// TIA Portal V20 export
// export: Created 2025-12-01T14:57:09.2054012Z, ExportSetting None, DisplayName Totally Integrated Automation Portal, DisplayVersion V20 Update 3, DisplayName TIA Portal Openness, DisplayVersion V20 Update 3, DisplayName TIA Portal Version Control Interface, DisplayVersion V20 Update 3, DisplayName STEP 7 Professional, DisplayVersion V20 Update 3, DisplayName STEP 7 Safety, DisplayVersion V20 Update 2, DisplayName WinCC Basic/Comfort/Advanced, DisplayVersion V20 Update 3, DisplayName WinCC Professional, DisplayVersion V20 Update 3, DisplayName WinCC Unified, DisplayVersion V20 Update 3
FUNCTION "FC834_GestorMaquinaSimple" : Void   // FC834, LAD
TITLE = Tracking de la Maquina Base
{ S7_Optimized_Access := 'FALSE' }
AUTHOR : TRACKING
NAME : 20160525
VERSION : 3.1
// - Inicializar
// - Recoger datos necesarios del Sistema
// 
// - Dispositivo Maquina
//   + Gestion de Estado
//   + Gestion de Control de Reset
//   + Gestion de Control de Paro Blando
//   + Gestion de Control de Errores
// 
// - Operaciones propias de la Maquina
// 
// - Cierre de protocolo de la Maquina
// - Actualizar datos del Sistema
// stored: AutoNumber false, SetENOAutomatically false
   VAR_INPUT
      DB_VIMaquina : DB_ANY;   // DB de la Maquina
      EstadoZonaMesa : "EstadoZona";   // Estado de la Zona Mesa Asociada a la Mesa
      NumMaquina : UInt;   // Numero de la Maquina
      RearmeError : Bool;   // Rearme de Errores Adicionales
      ManualReset : Bool;   // Resetear la Maquina desde el exterior
      FinReset : Bool;   // Reset Finalizado del VI Maquina
      ManualParoBlando : Bool;   // Paro Blando de la Mauina desde el exterior
      FinParoBlando : Bool;   // Paro Blando Finalizado del VI Maquina
   END_VAR
   VAR_TEMP
      PunteroDBVIMaquina : Any;
      P_EstadoVI : DWord;
      PunteroDBTMP : DWord;
      DBEstadoVI : Word;
      CodigoErrorMesa : UDInt;   // Error (Código) de la Mesa (Dispositivo)
      NumeroErrorVI : UInt;
      Maquina : UInt;   // Numero de Maquina dentro del PLC
      ByteTMP : Byte;
      ReturnValor : Int;
      TMPFinReset_NOK : Bool;
      TMPFinParoBlando_NOK : Bool;
      FlancoAuto : Bool;
      FlancoManual : Bool;
      FlancoMarcha : Bool;
      FlancoParo : Bool;
      FlancoReset : Bool;
      FlancoParoBlando : Bool;
      FinResetTMP : Bool;
      FinParoBlandoTMP : Bool;
   END_VAR
BEGIN

NETWORK
TITLE = Inicializar
/////////////////////////////////////////////////////////////////////////////
// --- Inicializar las Variables

      L     #NumMaquina;
      T     #Maquina;


/////////////////////////////////////////////////////////////////////////////
// --- Estado Mesa - Salida Inicializar a cero - Zona

      L     0;  // Que rellenar en el DB
      T     #ByteTMP;

      CALL  FILL
      ( BVAL    := #ByteTMP,
        RET_VAL := #ReturnValor,
        BLK     := "DB903_Estado_ZonaMaquina".EstadoMaquina[#Maquina]
      );  // Reseteo el la zona temp



NETWORK
TITLE = Gestion del Estado de la Maquina - Inicial
/////////////////////////////////////////////////////////////////////////////
// --- Flancos de los estados de la Maquina

      SET;
      A     #EstadoZonaMesa.Automatico_CBx;
      FP    "DB832_Maquinas".Maquinas[#Maquina].Memorias.MFL_Auto;  // Memo Automatico
      =     #FlancoAuto;

      SET;
      A     #EstadoZonaMesa.Manual_CBx;
      FP    "DB832_Maquinas".Maquinas[#Maquina].Memorias.MFL_Manual;  // Memo Manual
      =     #FlancoManual;

      SET;
      A     #EstadoZonaMesa.Marcha_CBx;
      FP    "DB832_Maquinas".Maquinas[#Maquina].Memorias.MFL_Marcha;  // Memo Marcha
      =     #FlancoMarcha;

      SET;
      A     #EstadoZonaMesa.Paro_CBx;
      FP    "DB832_Maquinas".Maquinas[#Maquina].Memorias.MFL_Paro;  // Memo Paro
      =     #FlancoParo;



NETWORK
TITLE = ---- Automatico, Manual
/////////////////////////////////////////////////////////////////////////////
// --- Estado de la Maquina
// --- Nota: Si cambia Auto/Remoto/Manual se pasa a Paro
// --- Nota: Si hay Marcha solo si esta en Automatico o Remoto
// ---       nunca en Manual

/////////////////////////////////////////////////////////////////////////////
// --- Maquina en Automatico (Estado: Automatico y Paro)
// --- Condicion: si la Zona Mesa esta en Automatico
      SET;
      A(;
      O     #FlancoAuto;  // Automatico de la Zona Mesa
      O     "DB841_Recepcion".DispoMaquina[#Maquina].Protocolo.Automatico;  // Automatico de la Orden Maquina
      );
      A     #EstadoZonaMesa.Automatico_CBx;  // Condicion
      JCN   NoEsta_EstadoDeLlaveEnAutomatico;

      SET;
      S     "DB840_Emision".DispoMaquina[#Maquina].Protocolo.Automatico;  // Poner en Automatico
      R     "DB840_Emision".DispoMaquina[#Maquina].Protocolo.Manual;

      JU    Final_EstadoDeLLave;

NoEsta_EstadoDeLlaveEnAutomatico:NOP   0;


/////////////////////////////////////////////////////////////////////////////
// --- Maquina en Manual (Estado: Manual y Paro)
// --- Condicion: Ninguna

      SET;
      A(;
      O     #FlancoManual;  // Manual de la Zona Mesa
      O     "DB841_Recepcion".DispoMaquina[#Maquina].Protocolo.Manual;  // Manual de la Orden Maquina
      );
      JCN   NoEsta_EstadoDeLlaveEnManual;

      SET;
      R     "DB840_Emision".DispoMaquina[#Maquina].Protocolo.Automatico;  // Poner en Manual
      S     "DB840_Emision".DispoMaquina[#Maquina].Protocolo.Manual;

      JU    Final_EstadoDeLLave;

NoEsta_EstadoDeLlaveEnManual:NOP   0;


/////////////////////////////////////////////////////////////////////////////
// --- Final Control de Llave de Mesa (En Automatico y En Manual)
Final_EstadoDeLLave:NOP   0;



NETWORK
TITLE = ---- Marcha, Paro
/////////////////////////////////////////////////////////////////////////////
// --- Maquina en Marcha
// --- Condicion: si esta la Maquina en Automatico o Remoto
// ---            si esta la Zona Mesa en Marcha

      SET;
      A(;
      O     #FlancoMarcha;  // Marcha de la Zona Mesa
      O     "DB841_Recepcion".DispoMaquina[#Maquina].Protocolo.Marcha;  // Marcha de la Orden Maquina
      );
      AN    #EstadoZonaMesa.Manual_CBx;  // Condiciones
      A     #EstadoZonaMesa.Marcha_CBx;

      AN    "DB840_Emision".DispoMaquina[#Maquina].Protocolo.Reset_Realizandose;
      JCN   NoEsta_EstadoDeMesaEnMarcha;

      SET;
      S     "DB840_Emision".DispoMaquina[#Maquina].Protocolo.Marcha;  // Poner en Marcha
      R     "DB840_Emision".DispoMaquina[#Maquina].Protocolo.Paro;
      R     "DB840_Emision".DispoMaquina[#Maquina].Protocolo.ParoBlando_Realizandose;  // Resetear Variables
      R     "DB840_Emision".DispoMaquina[#Maquina].Protocolo.ParoBlandoNOK;  // De Paro Blando
      R     "DB840_Emision".DispoMaquina[#Maquina].Protocolo.ParoBlandoOK;

      JU    Final_EstadoDeMesa;

NoEsta_EstadoDeMesaEnMarcha:NOP   0;


/////////////////////////////////////////////////////////////////////////////
// --- Maquina en Paro
// --- Condicion: Ninguna

      SET;
      A     #FlancoParo;  // Paro de la Zona Mesa
      O     "DB841_Recepcion".DispoMaquina[#Maquina].Protocolo.Paro;  // Paro de la Orden Maquina

      O     #FlancoAuto;  // Automatcio de la Zona Mesa
      O     #FlancoManual;  // Manual de la Zona Mesa

      O     "DB841_Recepcion".DispoMaquina[#Maquina].Protocolo.Automatico;  // Automatico de la Orden Maquina
      O     "DB841_Recepcion".DispoMaquina[#Maquina].Protocolo.Manual;  // Manual de la Orden Maquina

      JCN   NoEsta_EstadoDeMesaEnParo;

      SET;
      R     "DB840_Emision".DispoMaquina[#Maquina].Protocolo.Marcha;  // Poner en Paro
      S     "DB840_Emision".DispoMaquina[#Maquina].Protocolo.Paro;

NoEsta_EstadoDeMesaEnParo:NOP   0;


/////////////////////////////////////////////////////////////////////////////
// --- Final del control de Estado de Mesa (Marcha, Paro)
Final_EstadoDeMesa:NOP   0;




NETWORK
TITLE = Temporizador de Reset y Paro Blando NOK
/////////////////////////////////////////////////////////////////////////////
// --- Temporizador de Fin de Reset NOK

      CALL  "FC899_TMP"
      ( Temporizar     := "DB840_Emision".DispoMaquina[#Maquina].Protocolo.Reset_Realizandose,
        Valor_Tiempo   := "CTE_TMPEsperaFinReset",
        Base_tiempo_ms := 1000,
        Tiempo_OK      := #TMPFinReset_NOK,
        Valor_Actual   := "DB832_Maquinas".Maquinas[#Maquina].TMP_Reset
      );


/////////////////////////////////////////////////////////////////////////////
// --- Temporizador de Fin de ParoBlando NOK

      CALL  "FC899_TMP"
      ( Temporizar     := "DB840_Emision".DispoMaquina[#Maquina].Protocolo.ParoBlando_Realizandose,
        Valor_Tiempo   := "CTE_TMPEsperaFinReset",
        Base_tiempo_ms := 1000,
        Tiempo_OK      := #TMPFinParoBlando_NOK,
        Valor_Actual   := "DB832_Maquinas".Maquinas[#Maquina].TMP_ParoBlando
      );



NETWORK
TITLE = Gestion de Control de Reset
/////////////////////////////////////////////////////////////////////////////
// --- Flanco de Activacion de Reset

      SET;
      A     #EstadoZonaMesa.Resetear_CBx;  // Por la Zona Mesa
      O     #ManualReset;  // Manualmente (Exterior)
      O     "DB841_Recepcion".DispoMaquina[#Maquina].Protocolo.Reset;  // Por la Orden
      FP    "DB832_Maquinas".Maquinas[#Maquina].Memorias.MFL_Reset;  // Memo Reset
      =     #FlancoReset;

      SET;
      A     #FinReset;  // No hace caso si no hay Reset
      A     "DB904_Estado_Maquinas".EstadoVI[#Maquina].Fin_VI;
      A     "DB840_Emision".DispoMaquina[#Maquina].Protocolo.Reset_Realizandose;
      =     #FinResetTMP;

/////////////////////////////////////////////////////////////////////////////
// --- Activacion del Proceso de Reset

      SET;
      AN    #FlancoReset;
      JC    SistemaReset_Gestion;  // Hay que Realizar el Reset ?

      SET;
      A     "DB840_Emision".DispoMaquina[#Maquina].Protocolo.Marcha;
      JC    ResetImposible;


/////////////////////////////////////////////////////////////////////////////
// --- Se ha producido un Reset valido (Reseteo de las variables)

      SET;
      S     "DB840_Emision".DispoMaquina[#Maquina].Protocolo.Reset_Realizandose;  // Reseteando la Maquina
      R     "DB840_Emision".DispoMaquina[#Maquina].Protocolo.ParoBlando_Realizandose;  // Resetear Variables
      R     "DB840_Emision".DispoMaquina[#Maquina].Protocolo.ParoBlandoNOK;  // De Paro Blando
      R     "DB840_Emision".DispoMaquina[#Maquina].Protocolo.ParoBlandoOK;

      L     0;  // Reseteo el Status de Trabajo
      T     "DB832_Maquinas".Maquinas[#Maquina].MemoriaEstado;  // NuevoStatusTrabajo


/////////////////////////////////////////////////////////////////////////////
// --- Reseteo - DB del Vehiculo Inteligente

      OPN   #DB_VIMaquina;  // Abro el DB a resetear
      LAR1  P##PunteroDBVIMaquina;  // Preparar Puntero Any
      L     B#16#10;  // ID de Sintasis
      T     LB [AR1, P#0.0];
      L     B#16#2;  // Tipo de Datos
      T     LB [AR1, P#1.0];
      L     DBLG;  // Longitud del DB
      T     LW [AR1, P#2.0];
      L     DBNO;  // Numero de DB
      T     LW [AR1, P#4.0];
      L     0;
      SLW   3;
      T     LD [AR1, P#6.0];
      L     B#16#84;  // Indico el tipo DB
      T     LB [AR1, P#6.0];

      L     0;  // Que rellenar en el DB
      T     #ByteTMP;
      CALL  FILL
      ( BVAL    := #ByteTMP,
        RET_VAL := #ReturnValor,
        BLK     := #PunteroDBVIMaquina
      );  // Reseteo el DB


/////////////////////////////////////////////////////////////////////////////
// --- Reseteo - Estado del Vehiculo Inteligente

      L     0;  // Reseteo del Estado del VI
      T     #ByteTMP;
      CALL  FILL
      ( BVAL    := #ByteTMP,
        RET_VAL := #ReturnValor,
        BLK     := "DB904_Estado_Maquinas".EstadoVI[#Maquina]
      );


/////////////////////////////////////////////////////////////////////////////
// --- No hay más que resetar
      JU    SistemaReset_Gestion;


/////////////////////////////////////////////////////////////////////////////
// --- Reset Imposible

ResetImposible:NOP   0;
      SET;
      S     "DB840_Emision".DispoMaquina[#Maquina].Protocolo.ResetNOK;  // Activa del Bit Reset Imposible
      R     "DB840_Emision".DispoMaquina[#Maquina].Protocolo.ResetOK;  // Desactiva el Bit de Reset OK
      R     "DB840_Emision".DispoMaquina[#Maquina].Protocolo.Reset_Realizandose;

      JU    SistemaReset_Gestion;


/////////////////////////////////////////////////////////////////////////////
/////////////////////////////////////////////////////////////////////////////
/////////////////////////////////////////////////////////////////////////////
/////////////////////////////////////////////////////////////////////////////
// --- Gestion de Reset
SistemaReset_Gestion:NOP   0;
      SET;
      AN    "DB840_Emision".DispoMaquina[#Maquina].Protocolo.Reset_Realizandose;
      JC    SistemaReset_Fin;

      SET;
      AN    #EstadoZonaMesa.Resetear_CBx;  // Por la Zona
      AN    #EstadoZonaMesa.PerReset_CBx;
      AN    #ManualReset;  // Manualmente (Exterior)
      AN    "DB841_Recepcion".DispoMaquina[#Maquina].Protocolo.Reset;  // Por la Orden
      A     "DB841_Recepcion".DispoMaquina[#Maquina].Protocolo.EmiOK;  // Avisado el JdT ?
      JCN   SistemaReset_Continuar;


/////////////////////////////////////////////////////////////////////////////
// --- Reset Finalizazado
      SET;
      R     "DB840_Emision".DispoMaquina[#Maquina].Protocolo.Reset_Realizandose;


/////////////////////////////////////////////////////////////////////////////
// --- Continuar con el Reset
SistemaReset_Continuar:NOP   0;
      SET;
      A     #FinResetTMP;  // Fin de Reset del VI ?
      S     "DB840_Emision".DispoMaquina[#Maquina].Protocolo.ResetOK;  // Aviso de Fin de Reset


// --- Si no llega el Fin de Reset en un tiempo determinado
      SET;
      AN    #FinResetTMP;  // No, Fin de Reset del VI ?
      AN    "DB840_Emision".DispoMaquina[#Maquina].Protocolo.ResetOK;  // No, Aviso de Fin de Reset
      AN    "DB840_Emision".DispoMaquina[#Maquina].Protocolo.ResetNOK;  // No, Aviso de Fin de Reset
      A     #TMPFinReset_NOK;  // Se cumplido el tiempo de Espera
      A     "DB840_Emision".DispoMaquina[#Maquina].Protocolo.Reset_Realizandose;  // Reset Realizandose
      JC    ResetImposible;  // Activar reset imposible


/////////////////////////////////////////////////////////////////////////////
// --- Final de la Gestion de Reset
SistemaReset_Fin:NOP   0;
      SET;
      AN    "DB840_Emision".DispoMaquina[#Maquina].Protocolo.Reset_Realizandose;
      R     "DB840_Emision".DispoMaquina[#Maquina].Protocolo.ResetOK;  // No Aviso de Fin de Reset

      SET;
      A     "DB840_Emision".DispoMaquina[#Maquina].Protocolo.ResetNOK;
      A     "DB841_Recepcion".DispoMaquina[#Maquina].Protocolo.EmiOK;
      R     "DB840_Emision".DispoMaquina[#Maquina].Protocolo.ResetNOK;  // Desactivacion de Reset Imposible



NETWORK
TITLE = Gestion del Control de Paro Blando
// - Sistema de Paro Blando
//   * Flanco de Activacion del Paro Blando
//   * Activacion del proceso de Paro Blando
//   * Gestion del Paro Blando
/////////////////////////////////////////////////////////////////////////////
// --- Flanco de Activacion de Paro Blando

      SET;
      A     #EstadoZonaMesa.ParoBlando_CBx;  // Por la Zona Mesa
      O     #ManualParoBlando;  // Manualmente (Exterior)
      O     "DB841_Recepcion".DispoMaquina[#Maquina].Protocolo.ParoBlando;  // Por la Orden
      FP    "DB832_Maquinas".Maquinas[#Maquina].Memorias.MFL_ParoBlando;  // Memo Paro Blando - Pos: 22.7
      =     #FlancoParoBlando;

      SET;
      A     #FinParoBlando;  // No hace caso si no hay ParoBlando
      A     "DB904_Estado_Maquinas".EstadoVI[#Maquina].Paro_Blando;
      A     "DB840_Emision".DispoMaquina[#Maquina].Protocolo.ParoBlando_Realizandose;
      =     #FinParoBlandoTMP;


/////////////////////////////////////////////////////////////////////////////
// --- Activacion del Proceso de Paro Blando
      SET;
      AN    #FlancoParoBlando;
      JC    SistemaParoBlando_Gestion;  // Hay que Realizar el Paro Blando ?


/////////////////////////////////////////////////////////////////////////////
// --- Se ha producido un Paro Blando valido
      SET;
      S     "DB840_Emision".DispoMaquina[#Maquina].Protocolo.ParoBlando_Realizandose;  // Reseteando la Maquina

      JU    SistemaParoBlando_Gestion;


/////////////////////////////////////////////////////////////////////////////
// --- Paro Blando Imposible

ParoBlandoImposible:NOP   0;
      SET;
      S     "DB840_Emision".DispoMaquina[#Maquina].Protocolo.ParoBlandoNOK;  // Activacion de Paro Blando Imposible
      R     "DB840_Emision".DispoMaquina[#Maquina].Protocolo.ParoBlandoOK;  // DesActivacion de Paro Blando OK
      R     "DB840_Emision".DispoMaquina[#Maquina].Protocolo.ParoBlando_Realizandose;  // Acabado Paro Blando

      JU    SistemaParoBlando_Gestion;

/////////////////////////////////////////////////////////////////////////////
/////////////////////////////////////////////////////////////////////////////
/////////////////////////////////////////////////////////////////////////////
// --- Gestion de Paro Blando
SistemaParoBlando_Gestion:NOP   0;
      SET;
      AN    "DB840_Emision".DispoMaquina[#Maquina].Protocolo.ParoBlando_Realizandose;
      JC    SistemaParoBlando_Fin;

      SET;
      AN    #EstadoZonaMesa.ParoBlando_CBx;  // Por la Zona
      AN    #ManualParoBlando;  // Manualmente (Exterior)
      AN    "DB841_Recepcion".DispoMaquina[#Maquina].Protocolo.ParoBlando;  // Por la Orden
      A     "DB841_Recepcion".DispoMaquina[#Maquina].Protocolo.EmiOK;  // Avisado el JdT ?
      JCN   SistemaParoBlando_Continuar;


/////////////////////////////////////////////////////////////////////////////
/////////////////////////////////////////////////////////////////////////////
/////////////////////////////////////////////////////////////////////////////
// --- Paro Blando Finalizazado
      SET;
      R     "DB840_Emision".DispoMaquina[#Maquina].Protocolo.ParoBlando_Realizandose;


/////////////////////////////////////////////////////////////////////////////
/////////////////////////////////////////////////////////////////////////////
/////////////////////////////////////////////////////////////////////////////
// --- Continuar con el Reset
SistemaParoBlando_Continuar:NOP   0;
      SET;
      A     #FinParoBlandoTMP;  // Fin de Paro Blando del VI ?
      S     "DB840_Emision".DispoMaquina[#Maquina].Protocolo.ParoBlandoOK;  // Aviso de Fin de Paro Blando


// --- Si no llega el Fin de Paro Blando en un tiempo determinado
      SET;
      AN    #FinParoBlandoTMP;  // No, Fin de Paro Blando del VI ?
      AN    "DB840_Emision".DispoMaquina[#Maquina].Protocolo.ParoBlandoOK;  // No, Aviso de Fin de Paro Blando
      AN    "DB840_Emision".DispoMaquina[#Maquina].Protocolo.ParoBlandoNOK;  // No, Aviso de Fin de Paro Blando
      A     #TMPFinParoBlando_NOK;  // Se cumplido el tiempo de Espera
      A     "DB840_Emision".DispoMaquina[#Maquina].Protocolo.ParoBlando_Realizandose;  // Paro Blando Realizandose
      JC    ParoBlandoImposible;  // Activar Paro Blando imposible


/////////////////////////////////////////////////////////////////////////////
/////////////////////////////////////////////////////////////////////////////
/////////////////////////////////////////////////////////////////////////////
// --- Final de la Gestion de Reset
SistemaParoBlando_Fin:NOP   0;
      SET;
      AN    "DB840_Emision".DispoMaquina[#Maquina].Protocolo.ParoBlando_Realizandose;
      R     "DB840_Emision".DispoMaquina[#Maquina].Protocolo.ParoBlandoOK;  // No Aviso de Fin de Reset

      SET;
      A     "DB840_Emision".DispoMaquina[#Maquina].Protocolo.ParoBlandoNOK;
      A     "DB841_Recepcion".DispoMaquina[#Maquina].Protocolo.EmiOK;
      R     "DB840_Emision".DispoMaquina[#Maquina].Protocolo.ParoBlandoNOK;  // Desactivacion de Paro Blando Imposible



NETWORK
TITLE = Gestion de Control de Error de la Maquina
// - Calculo del Error de la Maquina
// - Rearme y Activacion del Error de la Maquina
/////////////////////////////////////////////////////////////////////////////
// --- Calculo del Error de la Mesa

      AN    "DB904_Estado_Maquinas".EstadoVI[#Maquina].Error_MAQx;
      JC    NoErrorEnMaquina;


/////////////////////////////////////////////////////////////////////////////
      L     #Maquina;  // Puntero al DB de Estado VI
      L     "CTE_Long_VIMaquina";  // Longitud de la UDT 20
      *D;
      SLD   3;
      T     #P_EstadoVI;

      L     "CTE_NDB_EstadoVIMaquina";  // DB de Estado VI
      T     #DBEstadoVI;

      L     #P_EstadoVI;  // Punteros
      L     P#2.0;
      +D;
      LAR2;
      T     #PunteroDBTMP;  // Offset dentro del DB

      OPN   DB [#DBEstadoVI];
Bucle_ErrorVI:NOP   0;
      A     DBX [AR2, P#0.0];
      JC    EncontradoErrorEnMaquina;

      +AR2  P#0.1;
      JU    Bucle_ErrorVI;


/////////////////////////////////////////////////////////////////////////////
// --- Con Error
EncontradoErrorEnMaquina:NOP   0;
      TAR2;
      L     #PunteroDBTMP;
      -D;
      L     51;
      +D;
      T     #NumeroErrorVI;
      T     "DB840_Emision".DispoMaquina[#Maquina].Error;

      L     #NumeroErrorVI;
      T     #CodigoErrorMesa;
      T     "DB861_FIFO_Errores".Maquinas[#Maquina];

      JU    FinGestion_Error;


/////////////////////////////////////////////////////////////////////////////
// --- Sin Error
NoErrorEnMaquina:NOP   0;
      L     0;
      T     #CodigoErrorMesa;
      T     "DB840_Emision".DispoMaquina[#Maquina].Error;
      T     "DB861_FIFO_Errores".Maquinas[#Maquina];

      JU    FinGestion_Error;


/////////////////////////////////////////////////////////////////////////////
// --- Rearme y Activacion del Error
FinGestion_Error:NOP   0;
      SET;
      A     #EstadoZonaMesa.Rearme_CBx;  // Por la Zona
      O     #RearmeError;  // Manualmente (Exterior)
      O     "DB841_Recepcion".DispoMaquina[#Maquina].Protocolo.Rearme;  // Por la Orden
      =     "DB903_Estado_ZonaMaquina".EstadoMaquina[#Maquina].Rearme_CBx;

      SET;
      A     "DB904_Estado_Maquinas".EstadoVI[#Maquina].Error_MAQx;
      =     "DB840_Emision".DispoMaquina[#Maquina].Protocolo.Error;  // Esta en Error el VI Maquina



REGION Network 9: Cierre del Protocolo de la Maquina
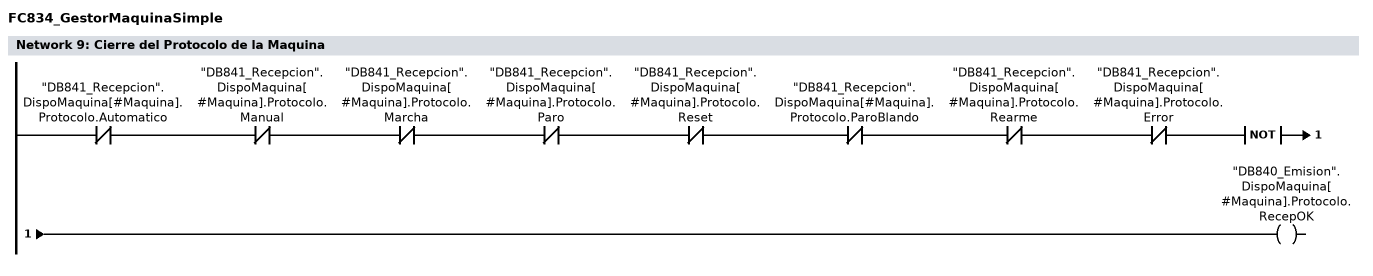
   RUNG wire#powerrail
      I_Contact( "DB841_Recepcion".DispoMaquina[#Maquina].Protocolo.Automatico )
      I_Contact( "DB841_Recepcion".DispoMaquina[#Maquina].Protocolo.Manual )
      I_Contact( "DB841_Recepcion".DispoMaquina[#Maquina].Protocolo.Marcha )
      I_Contact( "DB841_Recepcion".DispoMaquina[#Maquina].Protocolo.Paro )
      I_Contact( "DB841_Recepcion".DispoMaquina[#Maquina].Protocolo.Reset )
      I_Contact( "DB841_Recepcion".DispoMaquina[#Maquina].Protocolo.ParoBlando )
      I_Contact( "DB841_Recepcion".DispoMaquina[#Maquina].Protocolo.Rearme )
      I_Contact( "DB841_Recepcion".DispoMaquina[#Maquina].Protocolo.Error )
      Not()
      Coil( "DB840_Emision".DispoMaquina[#Maquina].Protocolo.RecepOK )
   END_RUNG
   // the same network as SCL:
   "DB840_Emision".DispoMaquina[#Maquina].Protocolo.RecepOK := NOT (NOT "DB841_Recepcion".DispoMaquina[#Maquina].Protocolo.Automatico AND NOT "DB841_Recepcion".DispoMaquina[#Maquina].Protocolo.Manual AND NOT "DB841_Recepcion".DispoMaquina[#Maquina].Protocolo.Marcha AND NOT "DB841_Recepcion".DispoMaquina[#Maquina].Protocolo.Paro AND NOT "DB841_Recepcion".DispoMaquina[#Maquina].Protocolo.Reset AND NOT "DB841_Recepcion".DispoMaquina[#Maquina].Protocolo.ParoBlando AND NOT "DB841_Recepcion".DispoMaquina[#Maquina].Protocolo.Rearme AND NOT "DB841_Recepcion".DispoMaquina[#Maquina].Protocolo.Error);
END_REGION

NETWORK
TITLE = Actualizacion del Estado para el Vehiculo Inteligente
/////////////////////////////////////////////////////////////////////////////
// --- Trasvase - Estado de la Maquina para VI

      A     "DB840_Emision".DispoMaquina[#Maquina].Protocolo.Error;
      =     "DB903_Estado_ZonaMaquina".EstadoMaquina[#Maquina].Error_CBx;
      A     "DB840_Emision".DispoMaquina[#Maquina].Protocolo.Marcha;
      =     "DB903_Estado_ZonaMaquina".EstadoMaquina[#Maquina].Marcha_CBx;
      A     "DB840_Emision".DispoMaquina[#Maquina].Protocolo.Paro;
      =     "DB903_Estado_ZonaMaquina".EstadoMaquina[#Maquina].Paro_CBx;

      A     "DB840_Emision".DispoMaquina[#Maquina].Protocolo.Automatico;
      =     "DB903_Estado_ZonaMaquina".EstadoMaquina[#Maquina].Automatico_CBx;
      A     "DB840_Emision".DispoMaquina[#Maquina].Protocolo.Manual;
      =     "DB903_Estado_ZonaMaquina".EstadoMaquina[#Maquina].Manual_CBx;

      A     #FlancoReset;
      =     "DB903_Estado_ZonaMaquina".EstadoMaquina[#Maquina].Resetear_CBx;
      A     "DB840_Emision".DispoMaquina[#Maquina].Protocolo.Reset_Realizandose;
      =     "DB903_Estado_ZonaMaquina".EstadoMaquina[#Maquina].PerReset_CBx;

      A     "DB840_Emision".DispoMaquina[#Maquina].Protocolo.ParoBlando_Realizandose;
      =     "DB903_Estado_ZonaMaquina".EstadoMaquina[#Maquina].ParoBlando_CBx;



NETWORK
TITLE = Introducir los Datos para el Scada
      CALL  "FC961_ScadaMaquina"
      ( NumMaquina := #Maquina
      );


END_FUNCTION
